ABB RAPID module: Part_2.mod

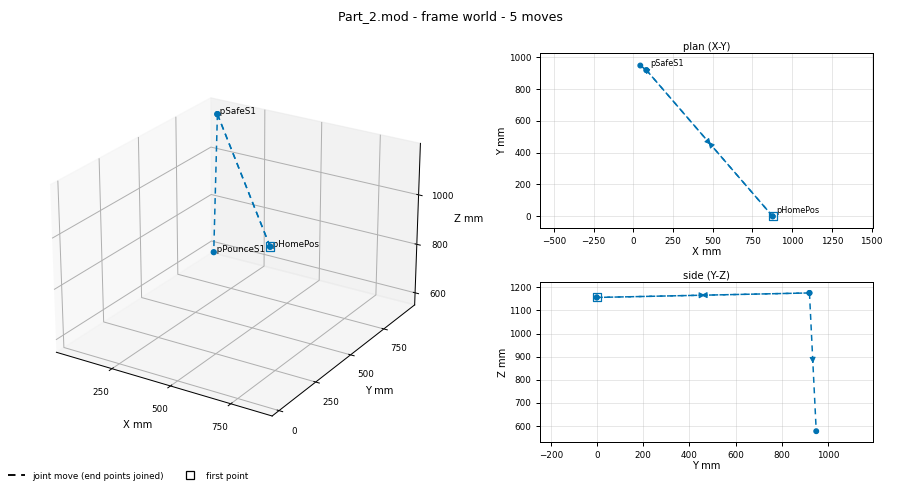
[picture p0: tool path of Part_2.mod in frame world, 5 of 13 moves have a stored position in this frame; points joined in program order, loops and branches not executed]
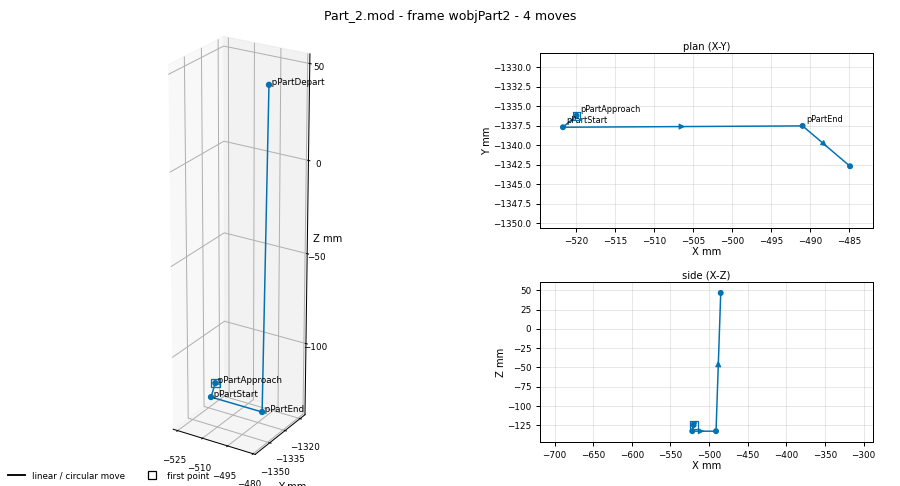
[picture p1: tool path of Part_2.mod in frame wobjPart2, 4 of 13 moves have a stored position in this frame; points joined in program order, loops and branches not executed]
MODULE Part_2
  ! ------------------------------------------------------------------
  ! Single-part welding template
  !
  ! Purpose:
  !   - Run one part only (no multi-part branching)
  !   - Keep nozzle cleaning and BullsEye tool check available
  !   - Provide a copy/paste starting point for new part files
  !
  ! Dependencies:
  !   - LogicZ (home/safe/pounce positions + rTC2013)
  !   - BE_User1 (BECheckToolb for BullsEye)
  !   - mTSC (optional torch cleaner if you prefer MechCleanGun)
  ! ------------------------------------------------------------------

  LOCAL PERS bool bUseTorchClean := TRUE;
  LOCAL PERS bool bUseBullseye := TRUE;

  ! Placeholder weld/seam data for the template. Replace with real values.
  LOCAL PERS welddata weldPart := [0,0,[1,0,0,0,0,0,0,0,0],[0,0,0,0,0,0,0,0,0]];
  LOCAL PERS seamdata seamPart := [1,1,[1,0,0,0,0,0,0,0,0],0,0,0,0,0,[0,0,0,0,0,0,0,0,0],0,0,[0,0,0,0,0,0,0,0,0],0,0,[0,0,0,0,0,0,0,0,0],0];

  ! Placeholder targets for the weld path. Replace with taught points.
  LOCAL CONST robtarget pPartApproach := [[-519.95,-1336.21,-124.59],[0.179682,0.6848,-0.680507,0.188877],[-2,-1,-3,0],[9E+09,9E+09,9E+09,9E+09,9E+09,9E+09]];
  CONST robtarget pPartStart := [[-521.69,-1337.70,-132.47],[0.193399,0.681112,-0.684086,0.175244],[-2,-1,-3,0],[9E+09,9E+09,9E+09,9E+09,9E+09,9E+09]];
  CONST robtarget pPartEnd := [[-490.93,-1337.53,-132.49],[0.193282,0.681205,-0.684029,0.175234],[-2,-1,-3,0],[9E+09,9E+09,9E+09,9E+09,9E+09,9E+09]];
  CONST robtarget pPartDepart := [[-484.84,-1342.71,46.50],[0.235633,0.655478,-0.679432,0.230648],[-2,-1,-3,0],[9E+09,9E+09,9E+09,9E+09,9E+09,9E+09]];
  PROC RunPart_2()
    TPWrite "Single-part template start";

    ! Optional BullsEye tool check before running a part.
    IF bUseBullseye THEN
      BECheckToolb;
    ENDIF

    ! Optional nozzle cleaning/reaming before the part weld.
    IF bUseTorchClean THEN
      rTC2013;
      ! Alternative: MechCleanGun;  ! From mTSC.mod
    ENDIF

    MoveJ pHomePos, v800, fine, tWeldGun;
    MoveJ pSafeS1, v800, fine, tWeldGun;
    MoveJ pPounceS1, v800, fine, tWeldGun;

    ! ----------------------------------------------------------------
    ! Single-part weld path (edit only the weld start/end points).
    ! ----------------------------------------------------------------
    IF bDryRun THEN
      MoveL DryRunTarget(pPartApproach), v200, z10, tWeldGun\WObj:=wobjPart2;
      MoveL DryRunTarget(pPartStart), v200, z10, tWeldGun\WObj:=wobjPart2;
      MoveL DryRunTarget(pPartEnd), v200, z10, tWeldGun\WObj:=wobjPart2;
      MoveL DryRunTarget(pPartDepart), v200, z10, tWeldGun\WObj:=wobjPart2;
    ELSE
      MoveL pPartApproach, v200, z10, tWeldGun\WObj:=wobjPart2;
      ArcLStart pPartStart, v30, seamPart, weldPart, fine, tWeldGun\WObj:=wobjPart2;
      ArcLEnd pPartEnd, v30, seamPart, weldPart, fine, tWeldGun\WObj:=wobjPart2;
      MoveL pPartDepart, v200, z10, tWeldGun\WObj:=wobjPart2;
    ENDIF

    MoveJ pSafeS1, v800, fine, tWeldGun;
    MoveJ pHomePos, v800, fine, tWeldGun;

    TPWrite "Single-part template complete";
  ENDPROC
ENDMODULE
